{attribute 'qualified_only'}
{attribute 'strict'}
{attribute 'to_string'}
TYPE E_DriveStates :
(
    INIT := 0,
    NO_FAULT := 1,
    SWITCH_ON_READY := 2,
    SWITCH_ON := 3,
    OPERATION_ENABLED := 4,
    FAULT := 5,
    FAULT_ACTIVE := 6,
    QUICK_STOP_ACTIVE := 7,
    MODE_ERROR := 8,
    WAIT	:= 9
) UINT;
END_TYPE

(* stored: Version 1.1.0.1
   DUT E_DriveStates: Id {81aaf441-a786-4eb3-9060-d17a0b007388} *)
